FUNCTION Camera_Set_Real : Buffer_Error
VAR_INPUT
	Camera : REFERENCE TO Cognex_Camera;
	Num : USINT;
	In : REAL;
END_VAR

Camera_Set_Real := Set_Real_From_Buffer(In:= In, 
										Num:= Num, 
										Layout:= Camera.Ouput_Buffer_Layout, 
										Buffer:= Camera.User_Data.UserData);

END_FUNCTION

(* stored: Version 1.1.0.1, ProductVersion 3.1.4024.10
   POU Camera_Set_Real: Id {92f652a1-f3d9-4f41-b78f-e3e3c96debd4}, SpecialFunc None *)
